# EPICS IOC start-up script: iocsh/ethercatmcslitAvoidCollSoftlimits.iocsh
dbLoadRecords("ethercatmcslitAvoidCollSoftlimits.template", "PREFIX=$(PREFIX), SLIT=$(SLIT), mXp=$(mXp), mXn=$(mXn) ")
